FUNCTION_BLOCK StackControl1 (* Basic Function Block Type *)
  (* Standard: 61499-2 *)
  (* Version 0.0, 9/29/2018, dmidro, nxtControl GmbH, Template *)
  PACKAGE Main;
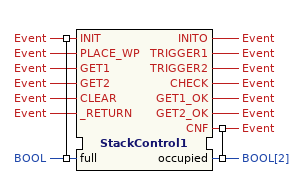
  EVENT_INPUT
    INIT WITH full; (* Initialization Request *)
    PLACE_WP; (* Normal Execution Request *)
    GET1;
    GET2;
    CLEAR;
    _RETURN;
  END_EVENT
  EVENT_OUTPUT
    INITO; (* Initialization Confirm *)
    TRIGGER1;
    TRIGGER2;
    CHECK;
    GET1_OK;
    GET2_OK;
    CNF WITH occupied; (* Execution Confirmation *)
  END_EVENT
  VAR_INPUT
    full : BOOL; (* Input event qualifier *)
  END_VAR
  VAR_OUTPUT
    occupied : ARRAY [0..1] OF BOOL;
  END_VAR
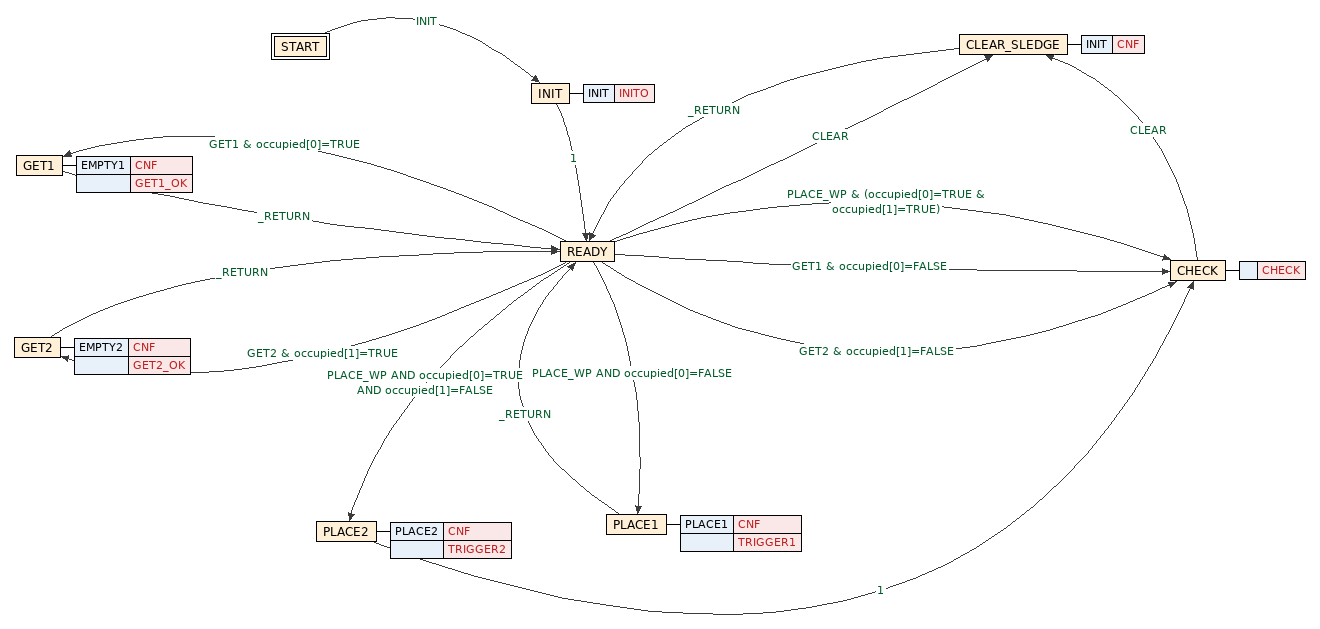
  EC_STATES
    START; (* Initial State *)
    INIT : INIT -> INITO; (* Initialization *)
    PLACE1 : PLACE1 -> CNF, -> TRIGGER1; (* Normal execution *)
    CHECK : -> CHECK;
    PLACE2 : PLACE2 -> CNF, -> TRIGGER2;
    GET1 : EMPTY1 -> CNF, -> GET1_OK;
    GET2 : EMPTY2 -> CNF, -> GET2_OK;
    READY;
    CLEAR_SLEDGE : INIT -> CNF;
  END_STATES
  EC_TRANSITIONS
    START TO INIT := INIT;
    INIT TO READY := 1;
    READY TO PLACE1 := PLACE_WP AND occupied[0]=FALSE;
    PLACE1 TO READY := _RETURN;
    READY TO CHECK := PLACE_WP & (occupied[0]=TRUE & occupied[1]=TRUE);
    READY TO CLEAR_SLEDGE := CLEAR;
    READY TO CHECK := GET1 & occupied[0]=FALSE;
    READY TO CHECK := GET2 & occupied[1]=FALSE;
    READY TO PLACE2 := PLACE_WP AND occupied[0]=TRUE AND occupied[1]=FALSE;
    PLACE2 TO CHECK := 1;
    READY TO GET1 := GET1 & occupied[0]=TRUE;
    GET1 TO READY := _RETURN;
    READY TO GET2 := GET2 & occupied[1]=TRUE;
    GET2 TO READY := _RETURN;
    CLEAR_SLEDGE TO READY := _RETURN;
    CHECK TO CLEAR_SLEDGE := CLEAR;
  END_TRANSITIONS
  ALGORITHM INIT IN ST: (* Initialization algorithm *)
;
IF full THEN
	occupied[0]:=TRUE;
	occupied[1]:=TRUE;
ELSE
	occupied[0]:=FALSE;
	occupied[1]:=FALSE;
END_IF;
  END_ALGORITHM
  ALGORITHM PLACE1 IN ST:
;
occupied[0]:=TRUE;
  END_ALGORITHM
  ALGORITHM PLACE2 IN ST:
;
occupied[1]:=TRUE;
  END_ALGORITHM
  ALGORITHM EMPTY1 IN ST:
;
occupied[0]:=FALSE;
  END_ALGORITHM
  ALGORITHM EMPTY2 IN ST:
;
occupied[1]:=FALSE;
  END_ALGORITHM
  ALGORITHM READY IN ST:
;
  END_ALGORITHM
END_FUNCTION_BLOCK
